# EPICS substitutions: danteApp/Db/dante1.substitutions
file "$(DANTE)/db/dante.template" {
{P=Dante:, R=dante1:, PORT=DANTE1, TRACE_LEN=16384}
}

file "$(DANTE)/db/danteN.template" {
{P=Dante:, R=dante1:, PORT=DANTE1, TRACE_LEN=16384}
}

file "$(DANTE)/db/dante1CH.template" {
{P=Dante:, R=dante1:, M=mca1, PORT=DANTE1}
}

file "$(MCA)/db/mca.db"
{
pattern
{   P,      M,       DTYP,         INP,         PREC,    NCHAN}
{Dante:,   mca1,  "asynMCA",  "@asyn(DANTE1,0)",   2,     4096}
}

file "$(ASYN)/db/asynRecord.db"
{
pattern
{P,             R,        PORT,   ADDR,  IMAX,  OMAX}
{Dante:, dante1:AsynIO, DANTE1,      0,    80,    80}
}
